(* CODESYS project WAGOIO v.1.0.0.library
   Version: 1.0.0.0
   Placeholder: WagoIO
   Title: WagoIO
   DocFormat: reStructuredText
   Company: Dicomat

Project tree, tasks and I/O mapping:
  Analog/
    function block AI_FLEX [ST]
    function AO_FLEX [ST]
  Doc/
*)

// Analog/AI_FLEX
(*

	ENTRADA ANALOGICA
		Si el móulo no está soportada se activa la alarma de instrumento y 
		el valor retornado es 999.99;
		Para los sensores temperatura tipo RTD y termopar se ignoran los
		parámetros de escalado a excepcion de los módulos  configurables como 
		el 750-451 ya que se	utilizan para la alarma de Sensor.
			
	Tarjetas Soportadas.
	=====================
		HART
			482 y 482001 (750-482/001) 

		0..20 mA
			452, 453, 465, 470
			480
			472

		4..20 mA, 
			454, 466, 455, 473
			485
			474

		RTD: No requieren configurar valores de Rango de escala.
			461, 481   --- 460
			451: No calcula error de sensor.

		Termopar: Si hay error de sensor retorn valor 0
			469: 2 canales
			458: 8 canales configurables. 

		NTC: 
			464020 (464/020)

		0..10v
			459, 467, 468, 477, 478, 497
			

	Valores de Salida:
			
	Control de Versiones:
	---------------------
	v2.12 04/03/2019
		* Corregido codigo 750-451. Esta referencia precisa definir
			la valores máximo y mínimo para generar la señal de error
			de lo contario esta estará activa continuamente. 
	
	v2.11 11/01/2019
		* Soporta Modulos HART: 750-482 y 750-482/001 (482001).

	v2.10 21/12/2018
		* Soporta Modulos 8 canales Entradas configurables de termopar 750-458.

	v2.9 01/07/2016
		* Soporta Modulos 8 canales Entradas configurables de Corriente 750-496.
		* Solamente esta soportados los modos de 0/4..20mA, NAMUR no esta soportado aún. 
	
	v2.8 01/07/2016
		* Soporta Modulos 8 canales Entradas configurables Tension  750-497

	v2.7 23/03/2016
		* Soport Modulos RTD configurable 750-451

	v2.6 10/07/2012
		* Modulos de pt100 cuando hay alarma de sensor el valor de salida es 0 en lugar de 850

	v2.4 10/07/2012
		* Se añade soporte tarjeta NTC 750-464/020-000 (464020)

*)
FUNCTION_BLOCK AI_FLEX
VAR_INPUT
	wRaw         : WORD;  (* Valor en bruto leido de la tarjeta analógica *)
	dwPartNumber : DWORD; (* Código Tarjeta Analógica  750-XXX*)
	rlMaxPV      : REAL;  (* Escalado de medida: Valor maximo de la  Variable de proceso *)
	rlMinPV      : REAL;  (* Escalado de medida: Valor Minimo  de la Variable de proceso *)
END_VAR

VAR_OUTPUT
	rlPV         : REAL;   (* Valor Calculado*)
	xError       : BOOL;  (* Error de Intrumento *)
END_VAR

VAR
	rlRaw         : REAL;
	rlMaxPVCount  : REAL;
END_VAR

xError:= FALSE;
CASE dwPartNumber OF
	451: (* Entradas de RTD Configurable*)
		rlPV:= INT_TO_REAL(wRaw) / 10.0;
		IF rlMaxPV = rlMinPV THEN
			xError:= TRUE; (* Alarma de Instrumento *)
		ELSE	
			IF rlPV >= rlMaxPV OR rlPV <= rlMinPV THEN
				xError:= TRUE; (* Alarma de Instrumento *)
			END_IF
		END_IF
		RETURN;

	452, 465, 470, 497: (* AI Medida 12 bits + 3 bits Status*)
		rlMaxPVCount:= WORD_TO_REAL(16#FFF); (*  *)
		IF (wRaw AND 16#01) <> 16#00 THEN
			xError:= TRUE; (* Alarma de Instrumento *)
		END_IF
		rlRaw:= SHR( wRaw, 3); (* Descarta bits de fuera de rango *)

	453: (* AI Entradas 0-20mA, Medida 12 bits + 3 bits Status*)
		rlMaxPVCount:= WORD_TO_REAL(16#FFF); (*  *)
		IF (wRaw AND 16#03) <> 16#00 THEN
			xError:= TRUE; (* Alarma de Instrumento *)
		END_IF
		rlRaw:= SHR( wRaw, 3); (* Descarta bits de fuera de rango *)

	454, 455, 466, 473: (* AI Entradas 4-20mA, Medida 12 bits + 3 bits Status*)
		rlMaxPVCount:= WORD_TO_REAL(16#FFF); (*  *)
		IF (wRaw AND 16#03) <> 16#00 THEN
			xError:= TRUE; (* Alarma de Instrumento *)
		END_IF
		rlRaw:= SHR( wRaw, 3); (* Descarta bits de fuera de rango *)

	472, 474, 478: (* AI Entradas 4-20mA y 0..10v: Medida 15 bits*)
		rlRaw:= wRaw;
		rlMaxPVCount:= WORD_TO_REAL(16#7FFF);

	460, 461, 481: (* AI type  RTD . supports All 750-461/xxx-xxx Models pt100 *)
		rlMaxPVCount:= 10.0;
		rlMaxPV:= 1;
		rlMinPV:= 0;
		rlRaw:= WORD_TO_INT(wRaw);
		IF (wRaw = 16#8001 OR wRaw = 8500) THEN
			xError:= TRUE; (* Alarma de Instrumento *)
			rlRaw:= 0;
		END_IF

	459, 468: (* AI Entradas 0..10v DC, Medida 12 bits + 3 bits Status*)
		rlMaxPVCount:= WORD_TO_REAL(16#FFF); (*  *)
		IF (wRaw AND 16#03) <> 16#00 THEN
			xError:= TRUE; (* Alarma de Instrumento *)
		END_IF
		rlRaw:= SHR( wRaw, 3); (* Descarta bits de fuera de rango *)

	464: (* Pt100 *)
		rlMaxPVCount:=10.0;
		rlMaxPV:= 1;
		rlMinPV:= 0;
		rlRaw:= INT_TO_REAL(WORD_TO_INT(wRaw));
		IF (wRaw = 16#F830) OR (wRaw = 16#2134)THEN
			xError:= TRUE; (* Alarma de Instrumento *)
			rlRaw:= 0;
		END_IF

	464020: (* NTC *)
		rlMaxPVCount:= 10.0;
		rlMaxPV:= 1;
		rlMinPV:= 0;
		rlRaw:= WORD_TO_INT(wRaw);
		IF rlRaw < -500.0 OR rlRaw > 1500 THEN
			xError:= TRUE; (* Alarma de Instrumento *)
		END_IF

	467, 477: (* AI Entradas 0-10v, Medida 16 bits*)
		rlRaw:= wRaw;
		rlMaxPVCount:= WORD_TO_REAL(16#FFFF);

	469, 458: (*  Termopar  *)
		rlMaxPVCount:= 10.0;
		rlMaxPV:= 1;
		rlMinPV:= 0;
		rlRaw:= INT_TO_REAL(WORD_TO_INT(wRaw));
		IF (wRaw = 16#07FFF) THEN
			xError:= TRUE; (* Alarma de Instrumento *)
			rlRaw:= 0;
		END_IF

	480: (* AI Entradas 0-20mA, Medida 13 bits + 2 bits Status*)
		rlMaxPVCount:= WORD_TO_REAL(16#1FFF); (*  *)
		IF (wRaw AND 16#03) <> 16#00 THEN
			xError:= TRUE; (* Alarma de Instrumento *)
		END_IF
		rlRaw:= SHR( wRaw, 2); (* Descarta bits de fuera de rango *)

	482: (* AI Entradas 4-20mA, Medida 12 bits + 2 bits Status*)
		rlMaxPVCount:= WORD_TO_REAL(16#1FFF); (*  *)
		IF (wRaw AND 16#03) <> 16#00 THEN
			xError:= TRUE; (* Alarma de Instrumento *)
		END_IF
		rlRaw:= SHR( wRaw, 2); (* Descarta bits de fuera de rango *)

	482001: (* AI Entradas 4-20mA, Medida 12 bits + 2 bits Status*)
		IF (wRaw AND 16#03) <> 16#00 THEN
			xError:= TRUE; (* Alarma de Instrumento *)
		END_IF
		rlMaxPVCount:= WORD_TO_REAL(7712); (*  *)
		rlRaw:= WORD_TO_INT(wRaw)/4; (* Descarta bits de fuera de rango *)

	485: (* AI Entradas 4-20mA, Medida 12 bits + 3 bits Status*)
		rlMaxPVCount:= INT_TO_REAL(16#FFF-819); (*  *)
		IF (wRaw AND 16#03) <> 16#00 THEN
			xError:= TRUE; (* Alarma de Instrumento *)
		END_IF
		rlRaw:= SHR( wRaw, 3)-819; (* Descarta bits de fuera de rango *)

	496: (* AI Entradas 4-20mA, Medida 12 bits + 3 bits Status*)
		rlMaxPVCount:= WORD_TO_REAL(16#FFF); (*  *)
		IF (wRaw AND 16#03) <> 16#00 THEN
			xError:= TRUE; (* Alarma de Instrumento *)
		END_IF
		rlRaw:= SHR( WORD_TO_INT(wRaw), 3); (* Descarta bits de fuera de rango *)

	ELSE
		xError:= TRUE; (* Alarma de Instrumento *)
		rlPV   := 999.99;
		RETURN;
END_CASE
rlPV:= (((rlMaxPV-rlMinPV)*rlRaw)/rlMaxPVCount)+ rlMinPV ; (* Cálculo en valor real *)

END_FUNCTION_BLOCK

// Analog/AO_FLEX
(******************************************************************************

	SALIDA ANALOGICA
		Si la tarjeta no está soportada el valor de salida es  0.
			
	Tarjetas Soportadas.
		0..20 mA
			552, 553

		4..20 mA
			554, 555
		
		0..10v
			550, 559
			
		-10v..+10v
			556, 557

		Configurables
			563, 597

			
	Control de Versiones:
	---------------------
	v2.3 01/07/2016
		* Soporta Modulos 8 canales Salidas configurables Tension 750-597

	v2.2 24/04/2015
		* Se añade tarjeta 750-563

	v2.1 09/04/2012
		* Se corrigen error de salida cunado el fondo de escala es ditinto de 0
		* Se añaden referencias a la lista de tarjeras soportadas.

	v2.0 23/04/2009
		* Versión Inicial


******************************************************************************)
FUNCTION AO_FLEX : WORD
VAR_INPUT
	rPV			: REAL;
	dwPartNumber	: DWORD;
	rMax			: REAL; (* MaxValue *)
	rMin			: REAL; (* *)
END_VAR
VAR
	rCardFullScale: REAL;
	factor: REAL;
END_VAR

AO_FLEX:= 0;
IF rPV > rMax THEN
	rPV:= rMax;
END_IF
IF rPV < rMin THEN
	rPV:= rMin;
END_IF

IF
	(dwPartNumber = 550) OR
	(dwPartNumber = 552) OR
	(dwPartNumber = 553) OR
	(dwPartNumber = 554) OR
	(dwPartNumber = 555) OR
	(dwPartNumber = 559) OR
	(dwPartNumber = 560) OR
	(dwPartNumber = 597) 	THEN (* 0..10v, 4..20mA 12Bits *)
	rCardFullScale:= 32767.0;
	AO_FLEX:= REAL_TO_WORD((rCardFullScale/(rMax - rMin)) * (rPV-rMin));
END_IF

IF	(dwPartNumber = 585) THEN (* 0..10v, 4..20mA 12Bits *)
	rCardFullScale:= 32767.0 - 6553;
	factor:= (rCardFullScale)/(rMax - rMin);
	AO_FLEX:= REAL_TO_WORD(factor * (rPV-rMin)) + (6553);
END_IF

IF	(dwPartNumber = 556) OR
	(dwPartNumber = 557) THEN (* -10..+10v  12Bits + signo *)
	rCardFullScale:= 65534.0;
	AO_FLEX:= REAL_TO_WORD((rCardFullScale/(rMax - rMin)) * (rPV-rMin)) - 32767;
END_IF

IF	(dwPartNumber = 563) THEN
	rCardFullScale:= 65535.0;
	AO_FLEX:= REAL_TO_WORD(((rCardFullScale/(rMax - rMin)) * (rPV-rMin)));
END_IF

END_FUNCTION
